Fanuc KAREL source: kb00024.KL

-- PROVISIONAL review KL for V940-1; original PC SHA256 dd83e23233cdce50cbe5ba9b788437e8199bb5d1966030e3a65484bf2ef067ca
-- Incomplete behavior may be omitted. Consult companion uncertainty JSON. Do not deploy.
PROGRAM KB00024
%NOLOCKGROUP
BEGIN
  -- V9_ZERO_TABLE_METADATA_HINT layout=0002_ascii; no indexed target words; source/name/runtime held
  -- UNRESOLVED_PC offsets 5-15; opcodes 27,22,31
  -- UNRESOLVED_PC offsets 20-24; opcodes 7F
END KB00024
